FUNCTION_BLOCK END_RUN_SEQ
VAR_INPUT
	xJigEndDone:		BOOL;
END_VAR
VAR_IN_OUT
	xExecute:			BOOL;
	xDone:				BOOL;
END_VAR
VAR_OUTPUT
END_VAR
VAR
	tpReset:			TP;
	rtDone:				R_TRIG;
	rtExecute:			R_TRIG;
	ftTimePulse:		F_TRIG;
	tpTimePulse:		TP;
	lrTargetPos:		LREAL;
	
	xTransCondition:	BOOL;	
	xTransRelease:		BOOL;
	SFCInit:			BOOL;
	SFCReset:			BOOL;	
	SFCError:			BOOL;
END_VAR

rtDone(CLK:=xDone);
IF rtDone.Q THEN
	xTransRelease:=FALSE;	
	SFCReset:=TRUE;
	xExecute:=FALSE;
END_IF

rtExecute(CLK:=xExecute);
IF rtExecute.Q THEN
	xTransRelease:=TRUE;
END_IF

aSEQ_ACT();

tpReset(IN:=SFCError, PT:=T#250MS);
SFCReset:= tpReset.Q;

ACTION ACK_DONE_AXIS_active:
IF G_sAxisDone.X OR G_sAxisDone.Y OR G_sAxisDone.Z OR G_sAxisDone.c THEN
	G_sAckAxisDone.X:=TRUE;
	G_sAckAxisDone.Y:=TRUE;
	G_sAckAxisDone.Z:=TRUE;
	G_sAckAxisDone.C:=TRUE;
ELSE
	G_sAckAxisDone.X:=FALSE;
	G_sAckAxisDone.Y:=FALSE;
	G_sAckAxisDone.Z:=FALSE;
	G_sAckAxisDone.C:=FALSE;
END_IF

xTransCondition:= NOT G_sAckAxisDone.X AND NOT G_sAckAxisDone.Y AND NOT G_sAckAxisDone.Z AND NOT G_sAckAxisDone.C;
END_ACTION

ACTION aSEQ_ACT:
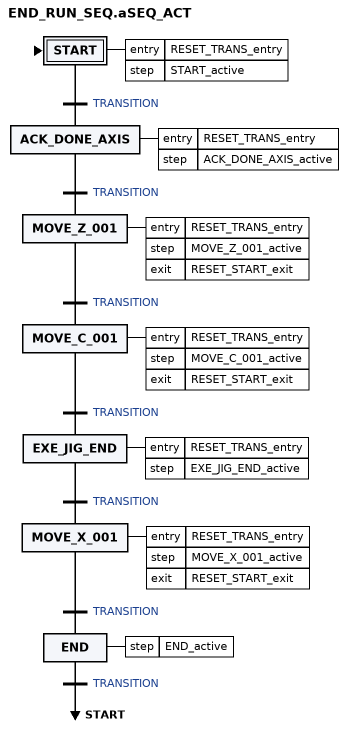
INITIAL_STEP START:
    RESET_TRANS_entry(P1);  // entry action
    START_active(N);  // step action
END_STEP
TRANSITION FROM START TO ACK_DONE_AXIS
    := TRANSITION;
END_TRANSITION
STEP ACK_DONE_AXIS:
    RESET_TRANS_entry(P1);  // entry action
    ACK_DONE_AXIS_active(N);  // step action
END_STEP
TRANSITION FROM ACK_DONE_AXIS TO MOVE_Z_001
    := TRANSITION;
END_TRANSITION
STEP MOVE_Z_001:
    RESET_TRANS_entry(P1);  // entry action
    MOVE_Z_001_active(N);  // step action
    RESET_START_exit(P0);  // exit action
END_STEP
TRANSITION FROM MOVE_Z_001 TO MOVE_C_001
    := TRANSITION;
END_TRANSITION
STEP MOVE_C_001:
    RESET_TRANS_entry(P1);  // entry action
    MOVE_C_001_active(N);  // step action
    RESET_START_exit(P0);  // exit action
END_STEP
TRANSITION FROM MOVE_C_001 TO EXE_JIG_END
    := TRANSITION;
END_TRANSITION
STEP EXE_JIG_END:
    RESET_TRANS_entry(P1);  // entry action
    EXE_JIG_END_active(N);  // step action
END_STEP
TRANSITION FROM EXE_JIG_END TO MOVE_X_001
    := TRANSITION;
END_TRANSITION
STEP MOVE_X_001:
    RESET_TRANS_entry(P1);  // entry action
    MOVE_X_001_active(N);  // step action
    RESET_START_exit(P0);  // exit action
END_STEP
TRANSITION FROM MOVE_X_001 TO END
    := TRANSITION;
END_TRANSITION
STEP END:
    END_active(N);  // step action
END_STEP
TRANSITION FROM END TO START
    := TRANSITION;
END_TRANSITION
END_ACTION

ACTION BLOW_DOWN_active:
tpTimePulse(IN:=NOT tpTimePulse.Q, PT:=T#3000MS);
ftTimePulse(CLK:=tpTimePulse.Q);
xTransCondition:= ftTimePulse.Q;
END_ACTION

ACTION END_active:
xDone:=TRUE;
xTransCondition:=xDone;
END_ACTION

ACTION EXE_JIG_END_active:
xTransCondition:=xJigEndDone;
END_ACTION

ACTION MOVE_C_001_active:
G_sControl.TargetPosition.C:= G_asIndividualAxisPositions[CE_AXIS_C].Positions[1].Target;
G_sStartToPos.C:= TRUE;

xTransCondition:= G_sAxisDone.C;
END_ACTION

ACTION MOVE_X_001_active:
G_sControl.TargetPosition.X:= G_asIndividualAxisPositions[CE_AXIS_X].Positions[1].Target;
G_sStartToPos.X:= TRUE;

xTransCondition:= G_sAxisDone.X;
END_ACTION

ACTION MOVE_Z_001_active:
G_sControl.TargetPosition.Z:= G_asIndividualAxisPositions[CE_AXIS_Z].Positions[1].Target;
G_sStartToPos.Z:= TRUE;

xTransCondition:= G_sAxisDone.Z;
END_ACTION

ACTION RESET_START_exit:
IF G_sAxisDone.X OR G_sAxisDone.Y OR G_sAxisDone.Z OR G_sAxisDone.c THEN
	G_sAckAxisDone.X:=TRUE;
	G_sAckAxisDone.Y:=TRUE;
	G_sAckAxisDone.Z:=TRUE;
	G_sAckAxisDone.C:=TRUE;
ELSE
	G_sAckAxisDone.X:=FALSE;
	G_sAckAxisDone.Y:=FALSE;
	G_sAckAxisDone.Z:=FALSE;
	G_sAckAxisDone.C:=FALSE;
	
	G_sStartToPos.X:=FALSE;
	G_sStartToPos.Y:=FALSE;
	G_sStartToPos.Z:=FALSE;
	G_sStartToPos.C:=FALSE;
END_IF
END_ACTION

ACTION RESET_TRANS_entry:
xTransCondition:= false;
END_ACTION

ACTION START_active:
xDone:=FALSE;
xTransCondition:= NOT xDone;
END_ACTION

TRANSITION TRANSITION:
xTransRelease AND xTransCondition
END_TRANSITION

END_FUNCTION_BLOCK

(* stored: Version 1.1.0.1, ProductVersion 3.1.4022.18
   POU END_RUN_SEQ: Id {bc6ad603-7798-4181-ad05-ef02a4f98eb2}, SpecialFunc None
   Folder xActive: Id {fba0e9d0-2437-4cd4-8919-34aeba4afa9a}
   Folder xEntry: Id {fdbc80b0-a244-4017-ad42-457e34fa86a3}
   Folder xExit: Id {a337dd26-7760-4f9b-8b6b-f06930d1b6f5}
   Folder xTrans: Id {eda636b8-71c9-43d1-b0e4-5bea8063b5c3}
   Action ACK_DONE_AXIS_active: Id {5df47b73-9d51-495f-8834-196c8ed521e1}
   Action aSEQ_ACT: Id {6e0df86b-1757-4ed9-b8f3-b63898deafee}
   Action BLOW_DOWN_active: Id {2311f086-c220-4506-9d3a-751abce7e4d1}
   Action END_active: Id {1f517bb0-1dc1-4788-be21-c812f57d6779}
   Action EXE_JIG_END_active: Id {4158d169-70f5-49c9-95bd-ffc06a364d40}
   Action MOVE_C_001_active: Id {5b08fe0d-dc14-4350-bd8b-d7ab183cf320}
   Action MOVE_X_001_active: Id {4ab2ff91-bc6d-4f66-858e-07bd1ea2a80f}
   Action MOVE_Z_001_active: Id {4838b9db-7888-4241-bfcb-76e00c0a82e1}
   Action RESET_START_exit: Id {11a9316e-b962-4042-8cb5-e47d4646a197}
   Action RESET_TRANS_entry: Id {5b7b4c24-8865-4986-9b2a-dfbab669e836}
   Action START_active: Id {529aba12-2b92-4708-bd3c-1bcd8d4b2490}
   Transition TRANSITION: Id {dadeedd2-126a-469f-b42b-32c4394085af} *)
